// TIA Portal V20 export
TYPE "Fuentes_Lineas"
   STRUCT
      Fuente : String[5];   // Nombre de la fuente
      Linea : Byte;   // Linea en la que esta conectada la tarjeta
      Posicion : Byte;   // posicion de la tarjeta en el cableado a partir de la fuente
   END_STRUCT;
END_TYPE
